INTERFACE I_Timer

PROPERTY Input : REFERENCE TO ST_Input
SET
END_SET
END_PROPERTY

PROPERTY Output : REFERENCE TO ST_Output
GET
END_GET
END_PROPERTY

METHOD Run
END_METHOD

PROPERTY Setting : REFERENCE TO ST_Setting
SET
END_SET
END_PROPERTY

END_INTERFACE

(* stored: Version 1.1.0.1, ProductVersion 3.1.4024.12
   Itf I_Timer: Id {c1c088be-f360-4e82-9631-f29e4a6f9dcb}
   Property Input: Id {30a681b4-13d2-46ce-90b2-2a29a995a827}
   Set Set: Id {5661becf-92b6-462f-9c38-91adfe6eb094}
   Property Output: Id {2330f76d-86bc-4fde-ba40-c3ea2ef5bd48}
   Get Get: Id {c56a5c12-5fe8-494b-9ba1-ed7e94e7952c}
   Method Run: Id {08ba81ea-83ed-47a5-bc9c-c0d88249effa}
   Property Setting: Id {72a2465f-006a-44f6-90e3-6c114dd71c8f}
   Set Set: Id {e40e6cae-f663-4d98-88d9-cf21a1218fb4} *)
